{attribute 'qualified_only'}
VAR_GLOBAL
END_VAR

(* stored: Version 1.1.0.1, ProductVersion 3.1.4022.18
   GVL COMM_GLV: Id {4863ef28-1f75-4073-a8c8-9ef85b85d696} *)
